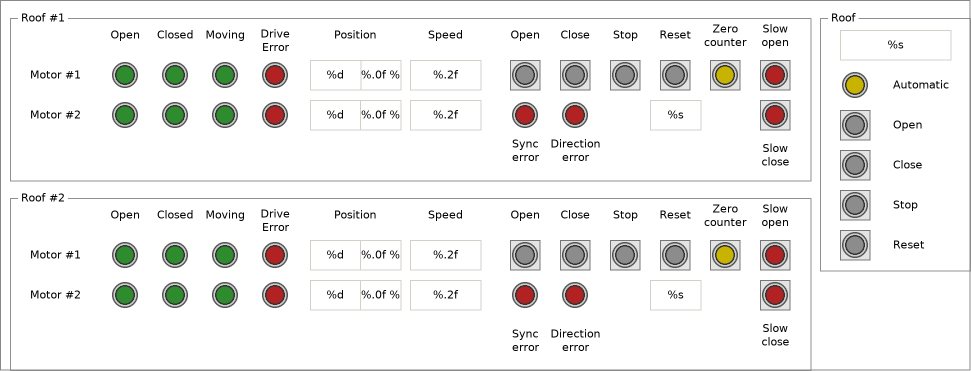
VISUALIZATION Roof  // 971x371
    GroupBox (10,10 801x171), "Roof #1"
        Label (10,50 71x30), "Motor #1"
        Label (10,90 71x30), "Motor #2"
        Label (80,10 71x30), "Open"
        Label (130,10 71x30), "Closed"
        Lamp1 (100,50 30x30), variable: MAIN.RoofControl.roofs[1].motors[1].opened, style: Lamp-Lamp1-Green
        Lamp1 (150,50 30x30), variable: MAIN.RoofControl.roofs[1].motors[1].closed, style: Lamp-Lamp1-Green
        Lamp1 (100,90 30x30), variable: MAIN.RoofControl.roofs[1].motors[2].opened, style: Lamp-Lamp1-Green
        Lamp1 (150,90 30x30), variable: MAIN.RoofControl.roofs[1].motors[2].closed, style: Lamp-Lamp1-Green
        Label (180,10 71x30), "Moving"
        Lamp1 (200,50 30x30), variable: MAIN.RoofControl.roofs[1].motors[1].moving, style: Lamp-Lamp1-Green
        Lamp1 (200,90 30x30), variable: MAIN.RoofControl.roofs[1].motors[2].moving, style: Lamp-Lamp1-Green
        Label (310,10 71x30), "Position"
        Textfield (350,50 41x30), "%.0f %", text variable: MAIN.RoofControl.roofs[1].motors[1].percent_open, input disabled if: TRUE
        Textfield (300,90 51x30), "%d", text variable: MAIN.RoofControl.roofs[1].motors[2].position, input disabled if: TRUE
        Label (400,10 71x30), "Speed"
        Textfield (400,50 71x30), "%.2f", text variable: MAIN.RoofControl.roofs[1].motors[1].speed, input disabled if: TRUE
        Textfield (400,90 71x30), "%.2f", text variable: MAIN.RoofControl.roofs[1].motors[2].speed, input disabled if: TRUE
        Label (480,10 71x30), "Open"
        PushSwitch (500,50 30x30), variable: MAIN.RoofControl.open_roof[1], behaviour: TAP, style: Switch-PushSwitch-Gray
        PushSwitch (550,50 30x30), variable: MAIN.RoofControl.close_roof[1], behaviour: TAP, style: Switch-PushSwitch-Gray
        Label (530,10 71x30), "Close"
        Label (590,10 51x30), "Stop"
        PushSwitch (600,50 30x30), variable: MAIN.RoofControl.stop_roof[1], behaviour: TAP, style: Switch-PushSwitch-Gray
        Lamp1 (500,90 30x30), variable: MAIN.RoofControl.roofs[1].sync_error, style: Lamp-Lamp1-Red
        Textfield (640,90 51x30), "%s", text variable: MAIN.RoofControl.roofs[1].state, input disabled if: TRUE
        Textfield (300,50 51x30), "%d", text variable: MAIN.RoofControl.roofs[1].motors[1].position, input disabled if: TRUE
        Textfield (350,90 41x30), "%.0f %", text variable: MAIN.RoofControl.roofs[1].motors[2].percent_open, input disabled if: TRUE
        Label (240,10 51x41), "Drive Error"
        Lamp1 (550,90 30x30), variable: MAIN.RoofControl.roofs[1].direction_error, style: Lamp-Lamp1-Red
        Label (490,120 51x41), "Sync error"
        Label (530,120 71x41), "Direction error"
        Label (640,10 51x30), "Reset"
        Lamp1 (250,50 30x30), variable: MAIN.RoofControl.roofs[1].motors[1].error, style: Lamp-Lamp1-Red
        Lamp1 (250,90 30x30), variable: MAIN.RoofControl.roofs[1].motors[2].error, style: Lamp-Lamp1-Red
        PushSwitch (750,50 30x30), variable: MAIN.RoofControl.roofs[1].slow_open, behaviour: TAP, style: Switch-PushSwitch-Red
        Label (740,10 51x31), "Slow open"
        Label (740,130 51x30), "Slow close"
        PushSwitch (750,230 30x30), variable: MAIN.RoofControl.stop_roof[1], behaviour: TAP, style: Switch-PushSwitch-Gray
        Label (690,10 51x31), "Zero counter"
    GroupBox (10,190 801x181), "Roof #2"
        Label (10,50 71x30), "Motor #1"
        Label (10,90 71x30), "Motor #2"
        Label (80,10 71x30), "Open"
        Label (130,10 71x30), "Closed"
        Lamp1 (100,50 30x30), variable: MAIN.RoofControl.roofs[2].motors[1].opened, style: Lamp-Lamp1-Green
        Lamp1 (150,50 30x30), variable: MAIN.RoofControl.roofs[2].motors[1].closed, style: Lamp-Lamp1-Green
        Lamp1 (100,90 30x30), variable: MAIN.RoofControl.roofs[2].motors[2].opened, style: Lamp-Lamp1-Green
        Lamp1 (150,90 30x30), variable: MAIN.RoofControl.roofs[2].motors[2].closed, style: Lamp-Lamp1-Green
        Label (180,10 71x30), "Moving"
        Lamp1 (200,50 30x30), variable: MAIN.RoofControl.roofs[2].motors[1].moving, style: Lamp-Lamp1-Green
        Lamp1 (200,90 30x30), variable: MAIN.RoofControl.roofs[2].motors[2].moving, style: Lamp-Lamp1-Green
        Label (310,10 71x30), "Position"
        Textfield (300,50 51x30), "%d", text variable: MAIN.RoofControl.roofs[2].motors[1].position, input disabled if: TRUE
        Textfield (300,90 51x30), "%d", text variable: MAIN.RoofControl.roofs[2].motors[2].position, input disabled if: TRUE
        Label (400,10 71x30), "Speed"
        Textfield (400,50 71x30), "%.2f", text variable: MAIN.RoofControl.roofs[2].motors[1].speed, input disabled if: TRUE
        Textfield (400,90 71x30), "%.2f", text variable: MAIN.RoofControl.roofs[2].motors[2].speed, input disabled if: TRUE
        Label (480,10 71x30), "Open"
        PushSwitch (500,50 30x30), variable: MAIN.RoofControl.open_roof[2], behaviour: TAP, style: Switch-PushSwitch-Gray
        PushSwitch (550,50 30x30), variable: MAIN.RoofControl.close_roof[2], behaviour: TAP, style: Switch-PushSwitch-Gray
        Label (530,10 71x30), "Close"
        Label (590,10 51x30), "Stop"
        PushSwitch (600,50 30x30), variable: MAIN.RoofControl.stop_roof[2], behaviour: TAP, style: Switch-PushSwitch-Gray
        Lamp1 (500,90 30x30), variable: MAIN.RoofControl.roofs[2].sync_error, style: Lamp-Lamp1-Red
        Textfield (640,90 51x30), "%s", text variable: MAIN.RoofControl.roofs[2].state, input disabled if: TRUE
        Textfield (350,50 41x30), "%.0f %", text variable: MAIN.RoofControl.roofs[2].motors[1].percent_open, input disabled if: TRUE
        Textfield (350,90 41x30), "%.0f %", text variable: MAIN.RoofControl.roofs[2].motors[2].percent_open, input disabled if: TRUE
        Label (240,10 51x41), "Drive Error"
        Label (490,130 51x41), "Sync error"
        Label (530,130 71x41), "Direction error"
        Lamp1 (550,90 30x30), variable: MAIN.RoofControl.roofs[2].direction_error, style: Lamp-Lamp1-Red
        Lamp1 (250,90 30x30), variable: MAIN.RoofControl.roofs[2].motors[2].error, style: Lamp-Lamp1-Red
        Lamp1 (250,50 30x30), variable: MAIN.RoofControl.roofs[2].motors[1].error, style: Lamp-Lamp1-Red
        PushSwitch (750,50 30x30), variable: MAIN.RoofControl.roofs[2].slow_open, behaviour: TAP, style: Switch-PushSwitch-Red
        PushSwitch (750,90 30x30), variable: MAIN.RoofControl.stop_roof[1], behaviour: TAP, style: Switch-PushSwitch-Gray
        PushSwitch (750,-90 30x30), variable: MAIN.RoofControl.stop_roof[1], behaviour: TAP, style: Switch-PushSwitch-Gray
        Label (740,130 51x30), "Slow close"
        Label (690,10 51x31), "Zero counter"
    GroupBox (820,10 151x261), "Roof"
        Label (70,100 71x30), "Open"
        PushSwitch (20,100 30x30), variable: MAIN.RoofControl.open_roofs, behaviour: TAP, style: Switch-PushSwitch-Gray
        PushSwitch (20,140 30x30), variable: MAIN.RoofControl.close_roofs, behaviour: TAP, style: Switch-PushSwitch-Gray
        Label (70,140 71x30), "Close"
        Label (70,180 71x30), "Stop"
        PushSwitch (20,180 30x30), variable: MAIN.RoofControl.stop_roofs, behaviour: TAP, style: Switch-PushSwitch-Gray
        Label (70,60 71x30), "Automatic"
        Lamp1 (20,60 30x30), variable: MAIN.RoofControl.automatic, style: Lamp-Lamp1-Yellow
        Label (70,220 71x30), "Reset"
        PushSwitch (20,220 30x30), variable: MAIN.RoofControl.reset_roofs, behaviour: TAP, style: Switch-PushSwitch-Gray
        Textfield (20,20 111x30), "%s", text variable: MAIN.RoofControl.roofs[1].state, input disabled if: TRUE
    PushSwitch (660,60 30x30), variable: MAIN.RoofControl.reset_roof[1], behaviour: TAP, style: Switch-PushSwitch-Gray
    Label (650,200 51x30), "Reset"
    PushSwitch (660,240 30x30), variable: MAIN.RoofControl.reset_roof[2], behaviour: TAP, style: Switch-PushSwitch-Gray
    PushSwitch (710,60 30x30), variable: MAIN.RoofControl.roofs[1].zero_counter, behaviour: TAP, style: Switch-PushSwitch-Yellow
    Label (750,200 51x31), "Slow open"
    PushSwitch (710,240 30x30), variable: MAIN.RoofControl.roofs[2].zero_counter, behaviour: TAP, style: Switch-PushSwitch-Yellow
    PushSwitch (760,280 30x30), variable: MAIN.RoofControl.roofs[2].slow_close, behaviour: TAP, style: Switch-PushSwitch-Red
    PushSwitch (760,100 30x30), variable: MAIN.RoofControl.roofs[1].slow_close, behaviour: TAP, style: Switch-PushSwitch-Red
END_VISUALIZATION

(* stored: Version 1.1.0.1, ProductVersion 3.1.4026.8
   Visu Roof: Id {e3a97d1b-e9a1-4ad0-8506-6ff5b42fdc2a} *)
